# EPICS substitutions: db/EL1098.substitutions
file EL1098.template
{ 	pattern
	{
		TERMINAL,
		DESC1,	ZNAM1,	ONAM1,	ZSV1,	OSV1,	COSV1,	SCAN1,
		DESC2,	ZNAM2,	ONAM2,	ZSV2,	OSV2,	COSV2,	SCAN2,
		DESC3,	ZNAM3,	ONAM3,	ZSV3,	OSV3,	COSV3,	SCAN3,
		DESC4,	ZNAM4,	ONAM4,	ZSV4,	OSV4,	COSV4,	SCAN4,
		DESC5,	ZNAM5,	ONAM5,	ZSV5,	OSV5,	COSV5,	SCAN5,
		DESC6,	ZNAM6,	ONAM6,	ZSV6,	OSV6,	COSV6,	SCAN6,
		DESC7,	ZNAM7,	ONAM7,	ZSV7,	OSV7,	COSV7,	SCAN7,
		DESC8,	ZNAM8,	ONAM8,	ZSV8,	OSV8,	COSV8,	SCAN8
	}
	{
	}
}
